{attribute addProperty BoxType "EP1859-0042-0018"}
{attribute addProperty Id "OutputAT %Q*BOOL81"}
{attribute addProperty CRC "2134331056"}
{attribute addProperty SizeInBites "8"}
{attribute addProperty SizeInBytes "1"}
TYPE DO_X05_Pin_7F374EB0 :
STRUCT
	{attribute addProperty Name "Output"}
	Output AT %Q* : BOOL;
END_STRUCT
END_TYPE

(* stored: Version 1.2.0.0, ProductVersion 3.1.4024.9
   DUT DO_X05_Pin_7F374EB0: Id {84e796ac-d9e6-4210-ae7b-a08aa1b4ac6e} *)
